// TIA Portal V20 export
// export: Created 2025-12-01T14:57:08.5037698Z, ExportSetting None, DisplayName Totally Integrated Automation Portal, DisplayVersion V20 Update 3, DisplayName TIA Portal Openness, DisplayVersion V20 Update 3, DisplayName TIA Portal Version Control Interface, DisplayVersion V20 Update 3, DisplayName STEP 7 Professional, DisplayVersion V20 Update 3, DisplayName STEP 7 Safety, DisplayVersion V20 Update 2, DisplayName WinCC Basic/Comfort/Advanced, DisplayVersion V20 Update 3, DisplayName WinCC Professional, DisplayVersion V20 Update 3, DisplayName WinCC Unified, DisplayVersion V20 Update 3
FUNCTION "FC983_CTRL_SmartMotor_3AD_1AT" : Void   // FC983, LAD
{ S7_Optimized_Access := 'TRUE' }
// stored: AutoNumber false, SetENOAutomatically false
   VAR_INPUT
      Avance : Bool;
      Retroceso_Manual : Bool;
      Vel_Rapida : Bool;
      Vel_Manual : Bool;
      T_Decel : UDInt;   // base tiempo ms
   END_VAR
   VAR_OUTPUT
      Av_Ret_Tx : Bool;
      DO1 : Bool;
      DO2 : Bool;
      DO3 : Bool;
   END_VAR
   VAR_IN_OUT
      TMP_Deceleracion : UDInt;
   END_VAR
   VAR_TEMP
      Parado_del_todo : Bool;
   END_VAR
BEGIN

REGION Network 1: Activación DI1 del Smart Motor
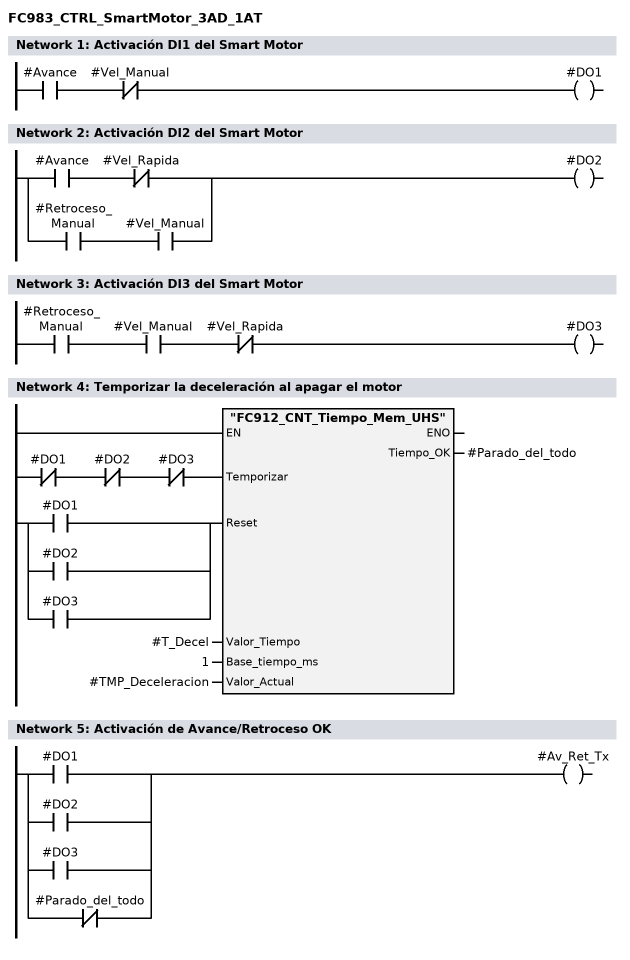
   RUNG wire#powerrail
      Contact( #Avance )
      I_Contact( #Vel_Manual )
      Coil( #DO1 )
   END_RUNG
   // the same network as SCL:
   #DO1 := #Avance AND NOT #Vel_Manual;
END_REGION

REGION Network 2: Activación DI2 del Smart Motor
   RUNG wire#powerrail
      Contact( #Avance )
      I_Contact( #Vel_Rapida )
      wire#w1
      Coil( #DO2 )
   END_RUNG
   RUNG wire#powerrail
      Contact( #Retroceso_Manual )
      Contact( #Vel_Manual )
   END_RUNG wire#w1
   // the same network as SCL:
   #DO2 := (#Avance AND NOT #Vel_Rapida) OR (#Retroceso_Manual AND #Vel_Manual);
END_REGION

REGION Network 3: Activación DI3 del Smart Motor
   RUNG wire#powerrail
      Contact( #Retroceso_Manual )
      Contact( #Vel_Manual )
      I_Contact( #Vel_Rapida )
      Coil( #DO3 )
   END_RUNG
   // the same network as SCL:
   #DO3 := #Retroceso_Manual AND #Vel_Manual AND NOT #Vel_Rapida;
END_REGION

REGION Network 4: Temporizar la deceleración al apagar el motor
   RUNG wire#powerrail
      "FC912_CNT_Tiempo_Mem_UHS"(Temporizar := wire#w1, Reset := wire#w2, Valor_Tiempo := #T_Decel, Base_tiempo_ms := 1, Valor_Actual := #TMP_Deceleracion, Tiempo_OK => #Parado_del_todo)
   END_RUNG
   RUNG wire#powerrail
      I_Contact( #DO1 )
      I_Contact( #DO2 )
      I_Contact( #DO3 )
   END_RUNG wire#w1
   RUNG wire#powerrail
      Contact( #DO1 )
   END_RUNG wire#w2
   RUNG wire#powerrail
      Contact( #DO2 )
   END_RUNG wire#w2
   RUNG wire#powerrail
      Contact( #DO3 )
   END_RUNG wire#w2
   // the same network as SCL:
   "FC912_CNT_Tiempo_Mem_UHS"(Temporizar := NOT #DO1 AND NOT #DO2 AND NOT #DO3,
                           Reset := #DO1 OR #DO2 OR #DO3,
                           Valor_Tiempo := #T_Decel,
                           Base_tiempo_ms := 1,
                           Valor_Actual := #TMP_Deceleracion,
                           Tiempo_OK => #Parado_del_todo);
END_REGION

REGION Network 5: Activación de Avance/Retroceso OK
   RUNG wire#powerrail
      Contact( #DO1 )
      wire#w1
      Coil( #Av_Ret_Tx )
   END_RUNG
   RUNG wire#powerrail
      Contact( #DO2 )
   END_RUNG wire#w1
   RUNG wire#powerrail
      Contact( #DO3 )
   END_RUNG wire#w1
   RUNG wire#powerrail
      I_Contact( #Parado_del_todo )
   END_RUNG wire#w1
   // the same network as SCL:
   #Av_Ret_Tx := #DO1 OR #DO2 OR #DO3 OR NOT #Parado_del_todo;
END_REGION
END_FUNCTION
